# EPICS autosave request: ADApp/Db/NDTransform_settings.req
$(P)$(R)Name
$(P)$(R)Type1
